// TIA Portal V20 export
// export: Created 2025-12-01T14:57:05.9594006Z, ExportSetting None, DisplayName Totally Integrated Automation Portal, DisplayVersion V20 Update 3, DisplayName TIA Portal Openness, DisplayVersion V20 Update 3, DisplayName TIA Portal Version Control Interface, DisplayVersion V20 Update 3, DisplayName STEP 7 Professional, DisplayVersion V20 Update 3, DisplayName STEP 7 Safety, DisplayVersion V20 Update 2, DisplayName WinCC Basic/Comfort/Advanced, DisplayVersion V20 Update 3, DisplayName WinCC Professional, DisplayVersion V20 Update 3, DisplayName WinCC Unified, DisplayVersion V20 Update 3
FUNCTION "FC899_TMP" : Void   // FC899, LAD
{ S7_Optimized_Access := 'FALSE' }
AUTHOR : TRACKING
NAME : 20150528
VERSION : 3.1
// stored: AutoNumber false, SetENOAutomatically false
   VAR_INPUT
      Temporizar : Bool;
      Valor_Tiempo : UDInt;
      Base_tiempo_ms : UDInt;
   END_VAR
   VAR_OUTPUT
      Tiempo_OK : Bool;
   END_VAR
   VAR_IN_OUT
      Valor_Actual : UDInt;
   END_VAR
   VAR_TEMP
      Aux_Inc_Tiempo : UDInt;
      TEMP_Tiempo_OK : Bool;
   END_VAR
BEGIN

REGION Network 1: ---
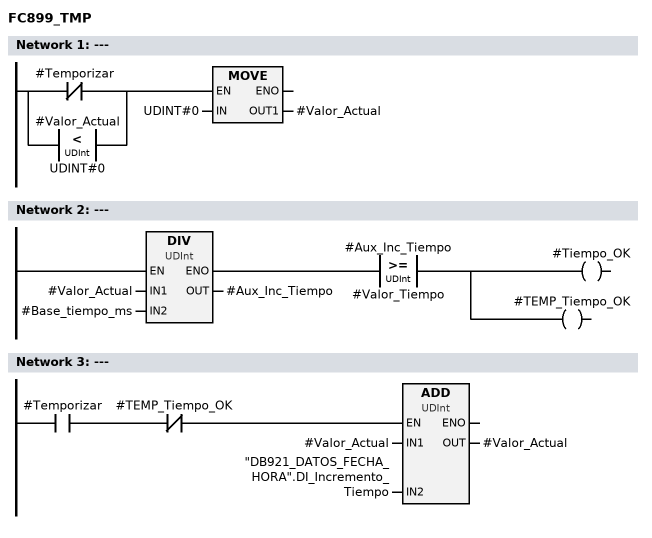
   RUNG wire#powerrail
      I_Contact( #Temporizar )
      wire#w1
      { S7_GenerateENO := "TRUE" } Move(in := UDINT#0, out1 => #Valor_Actual)
   END_RUNG
   RUNG wire#powerrail
      { S7_Templates := "SrcType := UDInt" } LT_Contact(in1 := #Valor_Actual, in2 := UDINT#0)
   END_RUNG wire#w1
   // the same network as SCL:
   IF NOT #Temporizar OR (#Valor_Actual < UDINT#0) THEN #Valor_Actual := UDINT#0; END_IF;
END_REGION

REGION Network 2: ---
   RUNG wire#powerrail
      { S7_Templates := "SrcType := UDInt"; S7_GenerateENO := "TRUE" } Div(in1 := #Valor_Actual, in2 := #Base_tiempo_ms, out => #Aux_Inc_Tiempo)
      { S7_Templates := "SrcType := UDInt" } GE_Contact(in1 := #Aux_Inc_Tiempo, in2 := #Valor_Tiempo)
      wire#w1
      Coil( #Tiempo_OK )
   END_RUNG
   RUNG wire#w1
      Coil( #TEMP_Tiempo_OK )
   END_RUNG
   // the same network as SCL:
   // ENO of a box is taken as its EN; it also drops when the box reports an error
   #Aux_Inc_Tiempo := #Valor_Actual / #Base_tiempo_ms;
   #Tiempo_OK := #Aux_Inc_Tiempo >= #Valor_Tiempo;
   #TEMP_Tiempo_OK := #Tiempo_OK;
END_REGION

REGION Network 3: ---
   RUNG wire#powerrail
      Contact( #Temporizar )
      I_Contact( #TEMP_Tiempo_OK )
      { S7_Templates := "SrcType := UDInt"; S7_GenerateENO := "TRUE" } Add(in1 := #Valor_Actual, in2 := "DB921_DATOS_FECHA_HORA".DI_Incremento_Tiempo, out => #Valor_Actual)
   END_RUNG
   // the same network as SCL:
   IF #Temporizar AND NOT #TEMP_Tiempo_OK THEN
       #Valor_Actual := #Valor_Actual + "DB921_DATOS_FECHA_HORA".DI_Incremento_Tiempo;
   END_IF;
END_REGION
END_FUNCTION
